INTERFACE itfContinuousAxisCommand EXTENDS itfAxisCommand

PROPERTY InVelocity : BOOL
GET
END_GET
END_PROPERTY

END_INTERFACE

(* stored: Version 1.1.0.1, ProductVersion 3.1.4024.11
   Itf itfContinuousAxisCommand: Id {b25e20ae-300b-47c7-9ad7-2fd307d32508}
   Property InVelocity: Id {e0a49328-fff5-44f5-bc83-800a8300e6c9}
   Get Get: Id {3fcdc4a1-ed9e-49f5-aba8-5b100cb2c880} *)
